// TIA Portal V18 export
FUNCTION "FC_DQ" : Void   // FC2, STL
{ S7_Optimized_Access := 'TRUE' }
VERSION : 0.1
// stored: AutoNumber true, UDAEnableTagReadback false
BEGIN

NETWORK
TITLE = 
      A     "DB_DQ".out_BeaconGreen;
      =     "out_BeaconGreen";

      A     "DB_DQ".out_BeaconRed;
      =     "out_BeaconRed";

      A     "DB_DQ".out_BeaconYellow;
      =     "out_BeaconYellow";

      A     "DB_DQ".out_GenPallet;
      =     "out_GenPallet";

      A     "DB_DQ".out_GenBox;
      =     "out_GenBox";

      A     "DB_DQ".out_5;
      =     "out_5";

      A     "DB_DQ".out_6;
      =     "out_6";

      A     "DB_DQ".out_7;
      =     "out_7";

      A     "DB_DQ".out_8;
      =     "out_8";

      A     "DB_DQ".out_Cov_0;
      =     "out_Cov_0";

      A     "DB_DQ".out_Cov_1;
      =     "out_Cov_1";

      A     "DB_DQ".out_Cov_1;
      =     "out_Cov_1";

      A     "DB_DQ".out_Cov_2;
      =     "out_Cov_2";

      A     "DB_DQ".out_Cov_3;
      =     "out_Cov_3";

      A     "DB_DQ".out_Cov_4;
      =     "out_Cov_4";

      A     "DB_DQ".out_Cov_5;
      =     "out_Cov_5";

      A     "DB_DQ".out_15;
      =     "out_15";

      A     "DB_DQ".out_Picker;
      =     "out_Picker";

      A     "DB_DQ".out_17;
      =     "out_17";

      A     "DB_DQ".out_18;
      =     "out_18";

      A     "DB_DQ".out_19;
      =     "out_19";

      A     "DB_DQ".out_20;
      =     "out_20";

      A     "DB_DQ".out_21;
      =     "out_21";

      A     "DB_DQ".out_22;
      =     "out_22";

      A     "DB_DQ".out_23;
      =     "out_23";

      A     "DB_DQ".out_BladesForward;
      =     "out_BladesFroward";

      A     "DB_DQ".out_BladesBackward;
      =     "out_BladesBackward";

      A     "DB_DQ".out_26;
      =     "out_26";

      A     "DB_DQ".out_27;
      =     "out_27";


















END_FUNCTION
